// TIA Portal project "仅数据块" (V17)

(* hardware
DEVICE "S7-1200 station_1"  S7-1200 Station
   slot 0: "Rack_0"  S7-1200 Rack  Rack  V1.0
   slot 1: "PLC_1"  CPU 1214C DC/DC/DC  6ES7 214-1AG40-0XB0  V4.2
*)

// ===== PLC "PLC_1"  CPU 1214C DC/DC/DC =====

VAR_GLOBAL   // PLC tag table "默认变量表"
   "Sensor1_Trigger" AT %I0.0 : Bool;   // 线圈
   "Sensor2_Trigger" AT %I0.1 : Bool;   // 线圈
   "Sensor3_Trigger" AT %I0.2 : Bool;   // 线圈
   "Camera_Ready" AT %I0.3 : Bool;   // 线圈
   "Camera_CaptureDone" AT %I0.4 : Bool;   // 线圈
   "Conv1_Run" AT %Q0.0 : Bool;   // 输出线圈
   "Conv2_Run" AT %Q0.1 : Bool;   // 输出线圈
   "Conv3_Run" AT %Q0.2 : Bool;   // 输出线圈
   "Conv4_Run" AT %Q0.3 : Bool;   // 输出线圈
   "Conv5_Run" AT %Q0.4 : Bool;   // 输出线圈
   "Camera_Trigger" AT %Q0.5 : Bool;   // 输出线圈
   "Indicator_Red" AT %Q0.6 : Bool;   // 输出线圈
   "Indicator_Green" AT %Q0.7 : Bool;   // 输出线圈
   "Indicator_Yellow" AT %Q1.0 : Bool;   // 输出线圈
   "System_Start" AT %Q1.1 : Bool;   // 输出线圈
   "System_Stop" AT %Q1.2 : Bool;   // 输出线圈
   "Tag_1" AT %M0.5 : Bool;
END_VAR

DATA_BLOCK "DB_AnalogCtrl"   // DB3
{ S7_Optimized_Access := 'FALSE' }
VERSION : 0.1
   VAR
      Conv1_SpeedSet : Int := 0;   // 寄存器
      Conv2_SpeedSet : Int;   // 寄存器
      Conv3_SpeedSet : Int;   // 寄存器
      Conv4_SpeedSet : Int;   // 寄存器
      Conv5_SpeedSet : Int;   // 寄存器
      Indicator_Status : Int;   // 寄存器
   END_VAR
BEGIN
END_DATA_BLOCK

DATA_BLOCK "CONNDB"   // DB5
{ S7_Optimized_Access := 'TRUE' }
VERSION : 0.1
   VAR
      CONN : TCON_IP_v4;
   END_VAR
BEGIN
   CONN.InterfaceId := 64;
   CONN.ID := 16#2;
   CONN.LocalPort := 502;
END_DATA_BLOCK

ORGANIZATION_BLOCK "Main"   // OB1, LAD, ProgramCycle
TITLE = "Main Program Sweep (Cycle)"
{ S7_Optimized_Access := 'TRUE' }
VERSION : 0.1
   VAR_INPUT
      Initial_Call : Bool;   // Initial call of this OB
      Remanence : Bool;   // =True, if remanent data are available
   END_VAR
BEGIN

REGION Network 1
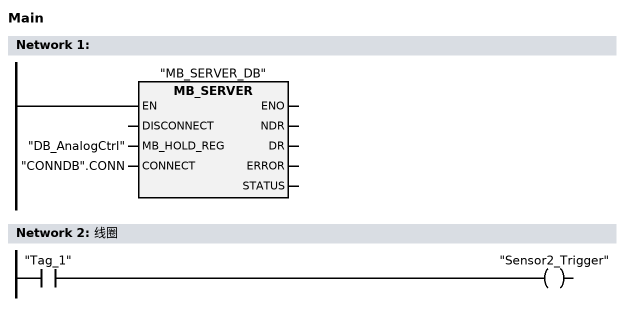
   "MB_SERVER_DB"(MB_HOLD_REG := "DB_AnalogCtrl", CONNECT := "CONNDB".CONN);   // MB_SERVER
END_REGION

REGION Network 2: 线圈
   RUNG wire#powerrail
      Contact( "Tag_1" )
      Coil( "Sensor2_Trigger" )
   END_RUNG
   // the same network as SCL:
   "Sensor2_Trigger" := "Tag_1";
END_REGION
END_ORGANIZATION_BLOCK